FUNCTION_BLOCK FB_InitializationSequence
VAR_INPUT
END_VAR
VAR_OUTPUT
END_VAR
VAR
END_VAR

END_FUNCTION_BLOCK

(* stored: Version 1.1.0.1, ProductVersion 3.1.4026.18
   POU FB_InitializationSequence: Id {e893420c-05db-404b-b76d-573468292b63}, SpecialFunc None *)
